			TT_01_01													:= m01_rs3_r3._01_TT_01,
			TT_01_01_offset												:= m01_rs3_r3.cart01_front_temp_offset,
			TT_01_01_error												:= m01_rs3_r3._01_TT_01_Error,
			TT_01_03													:= m01_rs3_r3._01_TT_03,               
			TT_01_03_offset												:= m01_rs3_r3.cart01_front_temp_offset,
			TT_01_03_error												:= m01_rs3_r3._01_TT_03_Error,         
			TT_02_01													:= m01_rs3_r3._02_TT_01,               
			TT_02_01_offset												:= m01_rs3_r3.cart02_front_temp_offset,
			TT_02_01_error												:= m01_rs3_r3._02_TT_01_Error,         
			TT_02_03													:= m01_rs3_r3._02_TT_03,               
			TT_02_03_offset												:= m01_rs3_r3.cart02_front_temp_offset,
			TT_02_03_error												:= m01_rs3_r3._02_TT_03_Error,         
			TT_03_01													:= m01_rs3_r3._03_TT_01,               
			TT_03_01_offset												:= m01_rs3_r3.cart03_front_temp_offset,
			TT_03_01_error												:= m01_rs3_r3._03_TT_01_Error,         
			TT_03_03													:= m01_rs3_r3._03_TT_03,               
			TT_03_03_offset												:= m01_rs3_r3.cart03_front_temp_offset,
			TT_03_03_error												:= m01_rs3_r3._03_TT_03_Error,         
			TT_04_01													:= m01_rs3_r3._04_TT_01,               
			TT_04_01_offset												:= m01_rs3_r3.cart04_front_temp_offset,
			TT_04_01_error												:= m01_rs3_r3._04_TT_01_Error,         
			TT_04_03													:= m01_rs3_r3._04_TT_03,               
			TT_04_03_offset												:= m01_rs3_r3.cart04_front_temp_offset,
			TT_04_03_error												:= m01_rs3_r3._04_TT_03_Error,         
			TT_05_01													:= m01_rs3_r3._05_TT_01,               
			TT_05_01_offset												:= m01_rs3_r3.cart05_front_temp_offset,
			TT_05_01_error												:= m01_rs3_r3._05_TT_01_Error,         
			TT_05_03													:= m01_rs3_r3._05_TT_03,               
			TT_05_03_offset												:= m01_rs3_r3.cart05_front_temp_offset,
			TT_05_03_error												:= m01_rs3_r3._05_TT_03_Error,         
			TT_06_01													:= m01_rs3_r3._06_TT_01,               
			TT_06_01_offset												:= m01_rs3_r3.cart06_front_temp_offset,
			TT_06_01_error												:= m01_rs3_r3._06_TT_01_Error,         
			TT_06_03													:= m01_rs3_r3._06_TT_03,               
			TT_06_03_offset												:= m01_rs3_r3.cart06_front_temp_offset,
			TT_06_03_error												:= m01_rs3_r3._06_TT_03_Error,         
			TT_07_01													:= m01_rs3_r3._07_TT_01,               
			TT_07_01_offset												:= m01_rs3_r3.cart07_front_temp_offset,
			TT_07_01_error												:= m01_rs3_r3._07_TT_01_Error,         
			TT_07_03													:= m01_rs3_r3._07_TT_03,               
			TT_07_03_offset												:= m01_rs3_r3.cart07_front_temp_offset,
			TT_07_03_error												:= m01_rs3_r3._07_TT_03_Error,         
			TT_08_01													:= m01_rs3_r3._08_TT_01,               
			TT_08_01_offset												:= m01_rs3_r3.cart08_front_temp_offset,
			TT_08_01_error												:= m01_rs3_r3._08_TT_01_Error,         
			TT_08_03													:= m01_rs3_r3._08_TT_03,               
			TT_08_03_offset												:= m01_rs3_r3.cart08_front_temp_offset,
			TT_08_03_error												:= m01_rs3_r3._08_TT_03_Error,         
			TT_09_01													:= m01_rs3_r3._09_TT_01,               
			TT_09_01_offset												:= m01_rs3_r3.cart09_front_temp_offset,
			TT_09_01_error												:= m01_rs3_r3._09_TT_01_Error,         
			TT_09_03													:= m01_rs3_r3._09_TT_03,               
			TT_09_03_offset												:= m01_rs3_r3.cart09_front_temp_offset,
			TT_09_03_error												:= m01_rs3_r3._09_TT_03_Error,         
			TT_10_01													:= m01_rs3_r3._10_TT_01,               
			TT_10_01_offset												:= m01_rs3_r3.cart10_front_temp_offset,
			TT_10_01_error												:= m01_rs3_r3._10_TT_01_Error,         
			TT_10_03													:= m01_rs3_r3._10_TT_03,               
			TT_10_03_offset												:= m01_rs3_r3.cart10_front_temp_offset,
			TT_10_03_error												:= m01_rs3_r3._10_TT_03_Error,         
			TT_11_01													:= m01_rs3_r3._11_TT_01,               
			TT_11_01_offset												:= m01_rs3_r3.cart11_front_temp_offset,
			TT_11_01_error												:= m01_rs3_r3._11_TT_01_Error,         
			TT_11_03													:= m01_rs3_r3._11_TT_03,               
			TT_11_03_offset												:= m01_rs3_r3.cart11_front_temp_offset,
			TT_11_03_error												:= m01_rs3_r3._11_TT_03_Error,         
			TT_12_01													:= m01_rs3_r3._12_TT_01,               
			TT_12_01_offset												:= m01_rs3_r3.cart12_front_temp_offset,
			TT_12_01_error												:= m01_rs3_r3._12_TT_01_Error,         
			TT_12_03													:= m01_rs3_r3._12_TT_03,               
			TT_12_03_offset												:= m01_rs3_r3.cart12_front_temp_offset,
			TT_12_03_error												:= m01_rs3_r3._12_TT_03_Error,         
		    
			cart01_front_temp											=> m01_rs3_r3.cart01_front_temp,						
			cart01_front_temp_error 									=> m01_rs3_r3.cart01_front_temp_error,
			cart01_back_temp											=> m01_rs3_r3.cart01_back_temp,
			cart01_back_temp_error 										=> m01_rs3_r3.cart01_back_temp_error,
			cart02_front_temp											=> m01_rs3_r3.cart02_front_temp,						
			cart02_front_temp_error 									=> m01_rs3_r3.cart02_front_temp_error,
			cart02_back_temp											=> m01_rs3_r3.cart02_back_temp,
			cart02_back_temp_error 										=> m01_rs3_r3.cart02_back_temp_error,
			cart03_front_temp											=> m01_rs3_r3.cart03_front_temp,						
			cart03_front_temp_error 									=> m01_rs3_r3.cart03_front_temp_error,
			cart03_back_temp											=> m01_rs3_r3.cart03_back_temp,
			cart03_back_temp_error 										=> m01_rs3_r3.cart03_back_temp_error,
			cart04_front_temp											=> m01_rs3_r3.cart04_front_temp,						
			cart04_front_temp_error 									=> m01_rs3_r3.cart04_front_temp_error,
			cart04_back_temp											=> m01_rs3_r3.cart04_back_temp,
			cart04_back_temp_error 										=> m01_rs3_r3.cart04_back_temp_error,
			cart05_front_temp											=> m01_rs3_r3.cart05_front_temp,						
			cart05_front_temp_error 									=> m01_rs3_r3.cart05_front_temp_error,
			cart05_back_temp											=> m01_rs3_r3.cart05_back_temp,
			cart05_back_temp_error 										=> m01_rs3_r3.cart05_back_temp_error,
			cart06_front_temp											=> m01_rs3_r3.cart06_front_temp,						
			cart06_front_temp_error 									=> m01_rs3_r3.cart06_front_temp_error,
			cart06_back_temp											=> m01_rs3_r3.cart06_back_temp,
			cart06_back_temp_error 										=> m01_rs3_r3.cart06_back_temp_error,
			cart07_front_temp											=> m01_rs3_r3.cart07_front_temp,						
			cart07_front_temp_error 									=> m01_rs3_r3.cart07_front_temp_error,
			cart07_back_temp											=> m01_rs3_r3.cart07_back_temp,
			cart07_back_temp_error 										=> m01_rs3_r3.cart07_back_temp_error,
			cart08_front_temp											=> m01_rs3_r3.cart08_front_temp,						
			cart08_front_temp_error 									=> m01_rs3_r3.cart08_front_temp_error,
			cart08_back_temp											=> m01_rs3_r3.cart08_back_temp,
			cart08_back_temp_error 										=> m01_rs3_r3.cart08_back_temp_error,
			cart09_front_temp											=> m01_rs3_r3.cart09_front_temp,						
			cart09_front_temp_error 									=> m01_rs3_r3.cart09_front_temp_error,
			cart09_back_temp											=> m01_rs3_r3.cart09_back_temp,
			cart09_back_temp_error 										=> m01_rs3_r3.cart09_back_temp_error,
			cart10_front_temp											=> m01_rs3_r3.cart10_front_temp,						
			cart10_front_temp_error 									=> m01_rs3_r3.cart10_front_temp_error,
			cart10_back_temp											=> m01_rs3_r3.cart10_back_temp,
			cart10_back_temp_error 										=> m01_rs3_r3.cart10_back_temp_error,
			cart11_front_temp											=> m01_rs3_r3.cart11_front_temp,						
			cart11_front_temp_error 									=> m01_rs3_r3.cart11_front_temp_error,
			cart11_back_temp											=> m01_rs3_r3.cart11_back_temp,
			cart11_back_temp_error 										=> m01_rs3_r3.cart11_back_temp_error,
			cart12_front_temp											=> m01_rs3_r3.cart12_front_temp,						
			cart12_front_temp_error 									=> m01_rs3_r3.cart12_front_temp_error,
			cart12_back_temp											=> m01_rs3_r3.cart12_back_temp,
			cart12_back_temp_error 										=> m01_rs3_r3.cart12_back_temp_error,    
                                                    
			inlet_co2_pump												:= m01_rs3_r3.inlet_co2_pump,
			AT_01_pump													=> m01_rs3_r3.AT_01_pump,
			inlet_co2_pump_cmd_status									=> m01_rs3_r3.inlet_co2_pump_cmd_status,
			inlet_co2_sol												:= m01_rs3_r3.inlet_co2_sol,
			AT_01_sol													=> m01_rs3_r3.AT_01_sol,
			inlet_co2_sol_cmd_status									=> m01_rs3_r3.inlet_co2_sol_cmd_status,
			outlet_co2_pump												:= m01_rs3_r3.outlet_co2_pump,
			AT_03_pump													=> m01_rs3_r3.AT_03_pump,
			outlet_co2_pump_cmd_status									=> m01_rs3_r3.outlet_co2_pump_cmd_status,
			outlet_co2_sol												:= m01_rs3_r3.outlet_co2_sol,
			AT_03_sol													=> m01_rs3_r3.AT_03_sol,
			outlet_co2_sol_cmd_status									=> m01_rs3_r3.outlet_co2_sol_cmd_status,
			repres_valve												:= m01_rs3_r3.repres_valve,
			XV_02														=> m01_rs3_r3.XV_02,
			repres_valve_open_cmd_status								=> m01_rs3_r3.repres_valve_open_cmd_status,
			repres_valve_open											:= m01_rs3_r3.repres_valve_open,
			repres_valve_closed											:= m01_rs3_r3.repres_valve_closed,
    	                                                        
			fan_vfd_control												=> m01_rs3_r3.fan_vfd_control,  		
			fan_vfd_target_vel	 		                                => m01_rs3_r3.fan_vfd_target_vel, 
			fan_vfd_enabled	 		                                    => m01_rs3_r3.fan_vfd_enabled, 
			fan_vfd_error		                                        => m01_rs3_r3.fan_vfd_error,
			fan_vfd_output												=> m01_rs3_r3.fan_vfd_output,
			fan_vfd_reset												:= m01_rs3_r3.fan_vfd_reset,
			fan_vfd_enable												:= m01_rs3_r3.fan_vfd_enable,
			fan_vfd_ecat_state											:= m01_rs3_r3.fan_vfd_ecat_state,
			fan_vfd_status												:= m01_rs3_r3.fan_vfd_status,
			fan_vfd														:= m01_rs3_r3.fan_vfd,
			fan_vfd_velocity											:= m01_rs3_r3.fan_vfd_velocity,
			fan_vfd_current												:= m01_rs3_r3.fan_vfd_current,
			fan_vfd_current_amps										=> m01_rs3_r3.fan_vfd_output_current,
			                                                    
			inlet_door_clamps_extend									:= m01_rs3_r3.inlet_door_clamps_extend,
			outlet_door_clamps_extend									:= m01_rs3_r3.outlet_door_clamps_extend,
			inlet_door_clamps_retract									:= m01_rs3_r3.inlet_door_clamps_retract,
			outlet_door_clamps_retract									:= m01_rs3_r3.outlet_door_clamps_retract,
			                                                    
			extend_clamps												:= extend_clamps,
			retract_clamps												:= retract_clamps,
			                                                    
			inlet_door_left_clamps_extend								=> m01_rs3_r3.XV_01_Left_Extend_Solenoid_Valve,
			inlet_door_right_clamps_extend								=> m01_rs3_r3.XV_01_Right_Extend_Solenoid_Valve,
			outlet_door_left_clamps_extend								=> m01_rs3_r3.XV_03_Left_Extend_Solenoid_Valve,
			outlet_door_right_clamps_extend								=> m01_rs3_r3.XV_03_Right_Extend_Solenoid_Valve,
			inlet_door_left_clamps_retract								=> m01_rs3_r3.XV_01_Left_Retract_Solenoid_Valve,
			inlet_door_right_clamps_retract								=> m01_rs3_r3.XV_01_Right_Retract_Solenoid_Valve,
			outlet_door_left_clamps_retract								=> m01_rs3_r3.XV_03_Left_Retract_Solenoid_Valve,
			outlet_door_right_clamps_retract							=> m01_rs3_r3.XV_03_Right_Retract_Solenoid_Valve,
    	                                                        
			inlet_door_left_clamps_extended								:= m01_rs3_r3.inlet_door_left_clamps_extended_ls,  
			inlet_door_right_clamps_extended							:= m01_rs3_r3.inlet_door_right_clamps_extended_ls, 
			outlet_door_left_clamps_extended							:= m01_rs3_r3.outlet_door_left_clamps_extended_ls, 
			outlet_door_right_clamps_extended							:= m01_rs3_r3.outlet_door_right_clamps_extended_ls,
			                                                    
			inlet_door_open												:= m01_rs3_r3.inlet_door_open,
			inlet_door_close											:= m01_rs3_r3.inlet_door_close,
			outlet_door_open											:= m01_rs3_r3.outlet_door_open,
			outlet_door_close											:= m01_rs3_r3.outlet_door_close,
			                                                    
			open_doors													:= open_doors,
			close_doors													:= close_doors,
			                                                    
			open_inlet_door												=> m01_rs3_r3.XV_01_Door_Open_Solenoid_Valve,
			close_inlet_door											=> m01_rs3_r3.XV_01_Door_Close_Solenoid_Valve,
			open_outlet_door											=> m01_rs3_r3.XV_03_Door_Open_Solenoid_Valve,
			close_outlet_door											=> m01_rs3_r3.XV_03_Door_Close_Solenoid_Valve,
			                                                    
			inlet_door_left_open										:= m01_rs3_r3.inlet_door_left_open_ls, 
			inlet_door_right_open										:= m01_rs3_r3.inlet_door_right_open_ls, 
			outlet_door_left_open										:= m01_rs3_r3.outlet_door_left_open_ls, 
			outlet_door_right_open										:= m01_rs3_r3.outlet_door_right_open_ls,
			inlet_door_left_closed										:= m01_rs3_r3.inlet_door_left_closed_ls, 
			inlet_door_right_closed										:= m01_rs3_r3.inlet_door_right_closed_ls, 
			outlet_door_left_closed										:= m01_rs3_r3.outlet_door_left_closed_ls, 
			outlet_door_right_closed									:= m01_rs3_r3.outlet_door_right_closed_ls,
			                                                    
			vacuum_cooling_high_temp_count								=> m01_rs3_r3.vacuum_cooling_high_temp_count,
			adsorption_high_temp_count									=> m01_rs3_r3.adsorption_high_temp_count,
			desorption_high_temp_count									=> m01_rs3_r3.desorption_air_high_temp_count);
END_ACTION

ACTION A_Reactor4_IO:
// Phase 0 - P_M01_RS03.A_Reactor4_IO
// Rev 1.0 - April 26, 2024

fb_R4_IO(	RSet														:= _RS03,
			React														:= _R4,
			
			Power_On													:= m01_rs3.power_control,
			                                                    
			sorbent_low_temp											=> m01_rs3_r4.temp_low,
			sorbent_high_temp											=> m01_rs3_r4.temp_high,
			sorbent_average_temp										=> m01_rs3_r4.temp_average,
			                                                    
			TT_01_01													:= m01_rs3_r4._01_TT_01,
			TT_01_01_offset												:= m01_rs3_r4.cart01_front_temp_offset,
			TT_01_01_error												:= m01_rs3_r4._01_TT_01_Error,
			TT_01_03													:= m01_rs3_r4._01_TT_03,               
			TT_01_03_offset												:= m01_rs3_r4.cart01_front_temp_offset,
			TT_01_03_error												:= m01_rs3_r4._01_TT_03_Error,         
			TT_02_01													:= m01_rs3_r4._02_TT_01,               
			TT_02_01_offset												:= m01_rs3_r4.cart02_front_temp_offset,
			TT_02_01_error												:= m01_rs3_r4._02_TT_01_Error,         
			TT_02_03													:= m01_rs3_r4._02_TT_03,               
			TT_02_03_offset												:= m01_rs3_r4.cart02_front_temp_offset,
			TT_02_03_error												:= m01_rs3_r4._02_TT_03_Error,         
			TT_03_01													:= m01_rs3_r4._03_TT_01,               
			TT_03_01_offset												:= m01_rs3_r4.cart03_front_temp_offset,
			TT_03_01_error												:= m01_rs3_r4._03_TT_01_Error,         
			TT_03_03													:= m01_rs3_r4._03_TT_03,               
			TT_03_03_offset												:= m01_rs3_r4.cart03_front_temp_offset,
			TT_03_03_error												:= m01_rs3_r4._03_TT_03_Error,         
			TT_04_01													:= m01_rs3_r4._04_TT_01,               
			TT_04_01_offset												:= m01_rs3_r4.cart04_front_temp_offset,
			TT_04_01_error												:= m01_rs3_r4._04_TT_01_Error,         
			TT_04_03													:= m01_rs3_r4._04_TT_03,               
			TT_04_03_offset												:= m01_rs3_r4.cart04_front_temp_offset,
			TT_04_03_error												:= m01_rs3_r4._04_TT_03_Error,         
			TT_05_01													:= m01_rs3_r4._05_TT_01,               
			TT_05_01_offset												:= m01_rs3_r4.cart05_front_temp_offset,
			TT_05_01_error												:= m01_rs3_r4._05_TT_01_Error,         
			TT_05_03													:= m01_rs3_r4._05_TT_03,               
			TT_05_03_offset												:= m01_rs3_r4.cart05_front_temp_offset,
			TT_05_03_error												:= m01_rs3_r4._05_TT_03_Error,         
			TT_06_01													:= m01_rs3_r4._06_TT_01,               
			TT_06_01_offset												:= m01_rs3_r4.cart06_front_temp_offset,
			TT_06_01_error												:= m01_rs3_r4._06_TT_01_Error,         
			TT_06_03													:= m01_rs3_r4._06_TT_03,               
			TT_06_03_offset												:= m01_rs3_r4.cart06_front_temp_offset,
			TT_06_03_error												:= m01_rs3_r4._06_TT_03_Error,         
			TT_07_01													:= m01_rs3_r4._07_TT_01,               
			TT_07_01_offset												:= m01_rs3_r4.cart07_front_temp_offset,
			TT_07_01_error												:= m01_rs3_r4._07_TT_01_Error,         
			TT_07_03													:= m01_rs3_r4._07_TT_03,               
			TT_07_03_offset												:= m01_rs3_r4.cart07_front_temp_offset,
			TT_07_03_error												:= m01_rs3_r4._07_TT_03_Error,         
			TT_08_01													:= m01_rs3_r4._08_TT_01,               
			TT_08_01_offset												:= m01_rs3_r4.cart08_front_temp_offset,
			TT_08_01_error												:= m01_rs3_r4._08_TT_01_Error,         
			TT_08_03													:= m01_rs3_r4._08_TT_03,               
			TT_08_03_offset												:= m01_rs3_r4.cart08_front_temp_offset,
			TT_08_03_error												:= m01_rs3_r4._08_TT_03_Error,         
			TT_09_01													:= m01_rs3_r4._09_TT_01,               
			TT_09_01_offset												:= m01_rs3_r4.cart09_front_temp_offset,
			TT_09_01_error												:= m01_rs3_r4._09_TT_01_Error,         
			TT_09_03													:= m01_rs3_r4._09_TT_03,               
			TT_09_03_offset												:= m01_rs3_r4.cart09_front_temp_offset,
			TT_09_03_error												:= m01_rs3_r4._09_TT_03_Error,         
			TT_10_01													:= m01_rs3_r4._10_TT_01,               
			TT_10_01_offset												:= m01_rs3_r4.cart10_front_temp_offset,
			TT_10_01_error												:= m01_rs3_r4._10_TT_01_Error,         
			TT_10_03													:= m01_rs3_r4._10_TT_03,               
			TT_10_03_offset												:= m01_rs3_r4.cart10_front_temp_offset,
			TT_10_03_error												:= m01_rs3_r4._10_TT_03_Error,         
			TT_11_01													:= m01_rs3_r4._11_TT_01,               
			TT_11_01_offset												:= m01_rs3_r4.cart11_front_temp_offset,
			TT_11_01_error												:= m01_rs3_r4._11_TT_01_Error,         
			TT_11_03													:= m01_rs3_r4._11_TT_03,               
			TT_11_03_offset												:= m01_rs3_r4.cart11_front_temp_offset,
			TT_11_03_error												:= m01_rs3_r4._11_TT_03_Error,         
			TT_12_01													:= m01_rs3_r4._12_TT_01,               
			TT_12_01_offset												:= m01_rs3_r4.cart12_front_temp_offset,
			TT_12_01_error												:= m01_rs3_r4._12_TT_01_Error,         
			TT_12_03													:= m01_rs3_r4._12_TT_03,               
			TT_12_03_offset												:= m01_rs3_r4.cart12_front_temp_offset,
			TT_12_03_error												:= m01_rs3_r4._12_TT_03_Error,         
		    
			cart01_front_temp											=> m01_rs3_r4.cart01_front_temp,						
			cart01_front_temp_error 									=> m01_rs3_r4.cart01_front_temp_error,
			cart01_back_temp											=> m01_rs3_r4.cart01_back_temp,
			cart01_back_temp_error 										=> m01_rs3_r4.cart01_back_temp_error,
			cart02_front_temp											=> m01_rs3_r4.cart02_front_temp,						
			cart02_front_temp_error 									=> m01_rs3_r4.cart02_front_temp_error,
			cart02_back_temp											=> m01_rs3_r4.cart02_back_temp,
			cart02_back_temp_error 										=> m01_rs3_r4.cart02_back_temp_error,
			cart03_front_temp											=> m01_rs3_r4.cart03_front_temp,						
			cart03_front_temp_error 									=> m01_rs3_r4.cart03_front_temp_error,
			cart03_back_temp											=> m01_rs3_r4.cart03_back_temp,
			cart03_back_temp_error 										=> m01_rs3_r4.cart03_back_temp_error,
			cart04_front_temp											=> m01_rs3_r4.cart04_front_temp,						
			cart04_front_temp_error 									=> m01_rs3_r4.cart04_front_temp_error,
			cart04_back_temp											=> m01_rs3_r4.cart04_back_temp,
			cart04_back_temp_error 										=> m01_rs3_r4.cart04_back_temp_error,
			cart05_front_temp											=> m01_rs3_r4.cart05_front_temp,						
			cart05_front_temp_error 									=> m01_rs3_r4.cart05_front_temp_error,
			cart05_back_temp											=> m01_rs3_r4.cart05_back_temp,
			cart05_back_temp_error 										=> m01_rs3_r4.cart05_back_temp_error,
			cart06_front_temp											=> m01_rs3_r4.cart06_front_temp,						
			cart06_front_temp_error 									=> m01_rs3_r4.cart06_front_temp_error,
			cart06_back_temp											=> m01_rs3_r4.cart06_back_temp,
			cart06_back_temp_error 										=> m01_rs3_r4.cart06_back_temp_error,
			cart07_front_temp											=> m01_rs3_r4.cart07_front_temp,						
			cart07_front_temp_error 									=> m01_rs3_r4.cart07_front_temp_error,
			cart07_back_temp											=> m01_rs3_r4.cart07_back_temp,
			cart07_back_temp_error 										=> m01_rs3_r4.cart07_back_temp_error,
			cart08_front_temp											=> m01_rs3_r4.cart08_front_temp,						
			cart08_front_temp_error 									=> m01_rs3_r4.cart08_front_temp_error,
			cart08_back_temp											=> m01_rs3_r4.cart08_back_temp,
			cart08_back_temp_error 										=> m01_rs3_r4.cart08_back_temp_error,
			cart09_front_temp											=> m01_rs3_r4.cart09_front_temp,						
			cart09_front_temp_error 									=> m01_rs3_r4.cart09_front_temp_error,
			cart09_back_temp											=> m01_rs3_r4.cart09_back_temp,
			cart09_back_temp_error 										=> m01_rs3_r4.cart09_back_temp_error,
			cart10_front_temp											=> m01_rs3_r4.cart10_front_temp,						
			cart10_front_temp_error 									=> m01_rs3_r4.cart10_front_temp_error,
			cart10_back_temp											=> m01_rs3_r4.cart10_back_temp,
			cart10_back_temp_error 										=> m01_rs3_r4.cart10_back_temp_error,
			cart11_front_temp											=> m01_rs3_r4.cart11_front_temp,						
			cart11_front_temp_error 									=> m01_rs3_r4.cart11_front_temp_error,
			cart11_back_temp											=> m01_rs3_r4.cart11_back_temp,
			cart11_back_temp_error 										=> m01_rs3_r4.cart11_back_temp_error,
			cart12_front_temp											=> m01_rs3_r4.cart12_front_temp,						
			cart12_front_temp_error 									=> m01_rs3_r4.cart12_front_temp_error,
			cart12_back_temp											=> m01_rs3_r4.cart12_back_temp,
			cart12_back_temp_error 										=> m01_rs3_r4.cart12_back_temp_error,  

                                                    
			inlet_co2_pump												:= m01_rs3_r4.inlet_co2_pump,
			AT_01_pump													=> m01_rs3_r4.AT_01_pump,
			inlet_co2_pump_cmd_status									=> m01_rs3_r4.inlet_co2_pump_cmd_status,
			inlet_co2_sol												:= m01_rs3_r4.inlet_co2_sol,
			AT_01_sol													=> m01_rs3_r4.AT_01_sol,
			inlet_co2_sol_cmd_status									=> m01_rs3_r4.inlet_co2_sol_cmd_status,
			outlet_co2_pump												:= m01_rs3_r4.outlet_co2_pump,
			AT_03_pump													=> m01_rs3_r4.AT_03_pump,
			outlet_co2_pump_cmd_status									=> m01_rs3_r4.outlet_co2_pump_cmd_status,
			outlet_co2_sol												:= m01_rs3_r4.outlet_co2_sol,
			AT_03_sol													=> m01_rs3_r4.AT_03_sol,
			outlet_co2_sol_cmd_status									=> m01_rs3_r4.outlet_co2_sol_cmd_status,
			repres_valve												:= m01_rs3_r4.repres_valve,
			XV_02														=> m01_rs3_r4.XV_02,
			repres_valve_open_cmd_status								=> m01_rs3_r4.repres_valve_open_cmd_status,
			repres_valve_open											:= m01_rs3_r4.repres_valve_open,
			repres_valve_closed											:= m01_rs3_r4.repres_valve_closed,
    	                                                        
			fan_vfd_control												=> m01_rs3_r4.fan_vfd_control,  		
			fan_vfd_target_vel	 		                                => m01_rs3_r4.fan_vfd_target_vel, 
			fan_vfd_enabled	 		                                    => m01_rs3_r4.fan_vfd_enabled, 
			fan_vfd_error		                                        => m01_rs3_r4.fan_vfd_error,
			fan_vfd_output												=> m01_rs3_r4.fan_vfd_output,
			fan_vfd_reset												:= m01_rs3_r4.fan_vfd_reset,
			fan_vfd_enable												:= m01_rs3_r4.fan_vfd_enable,
			fan_vfd_ecat_state											:= m01_rs3_r4.fan_vfd_ecat_state,
			fan_vfd_status												:= m01_rs3_r4.fan_vfd_status,
			fan_vfd														:= m01_rs3_r4.fan_vfd,
			fan_vfd_velocity											:= m01_rs3_r4.fan_vfd_velocity,
			fan_vfd_current												:= m01_rs3_r4.fan_vfd_current,
			fan_vfd_current_amps										=> m01_rs3_r4.fan_vfd_output_current,
			                                                    
			inlet_door_clamps_extend									:= m01_rs3_r4.inlet_door_clamps_extend,
			outlet_door_clamps_extend									:= m01_rs3_r4.outlet_door_clamps_extend,
			inlet_door_clamps_retract									:= m01_rs3_r4.inlet_door_clamps_retract,
			outlet_door_clamps_retract									:= m01_rs3_r4.outlet_door_clamps_retract,
			                                                    
			extend_clamps												:= extend_clamps,
			retract_clamps												:= retract_clamps,
			                                                    
			inlet_door_left_clamps_extend								=> m01_rs3_r4.XV_01_Left_Extend_Solenoid_Valve,
			inlet_door_right_clamps_extend								=> m01_rs3_r4.XV_01_Right_Extend_Solenoid_Valve,
			outlet_door_left_clamps_extend								=> m01_rs3_r4.XV_03_Left_Extend_Solenoid_Valve,
			outlet_door_right_clamps_extend								=> m01_rs3_r4.XV_03_Right_Extend_Solenoid_Valve,
			inlet_door_left_clamps_retract								=> m01_rs3_r4.XV_01_Left_Retract_Solenoid_Valve,
			inlet_door_right_clamps_retract								=> m01_rs3_r4.XV_01_Right_Retract_Solenoid_Valve,
			outlet_door_left_clamps_retract								=> m01_rs3_r4.XV_03_Left_Retract_Solenoid_Valve,
			outlet_door_right_clamps_retract							=> m01_rs3_r4.XV_03_Right_Retract_Solenoid_Valve,
    	                                                        
			inlet_door_left_clamps_extended								:= m01_rs3_r4.inlet_door_left_clamps_extended_ls,  
			inlet_door_right_clamps_extended							:= m01_rs3_r4.inlet_door_right_clamps_extended_ls, 
			outlet_door_left_clamps_extended							:= m01_rs3_r4.outlet_door_left_clamps_extended_ls, 
			outlet_door_right_clamps_extended							:= m01_rs3_r4.outlet_door_right_clamps_extended_ls,
			                                                    
			inlet_door_open												:= m01_rs3_r4.inlet_door_open,
			inlet_door_close											:= m01_rs3_r4.inlet_door_close,
			outlet_door_open											:= m01_rs3_r4.outlet_door_open,
			outlet_door_close											:= m01_rs3_r4.outlet_door_close,
			                                                    
			open_doors													:= open_doors,
			close_doors													:= close_doors,
			                                                    
			open_inlet_door												=> m01_rs3_r4.XV_01_Door_Open_Solenoid_Valve,
			close_inlet_door											=> m01_rs3_r4.XV_01_Door_Close_Solenoid_Valve,
			open_outlet_door											=> m01_rs3_r4.XV_03_Door_Open_Solenoid_Valve,
			close_outlet_door											=> m01_rs3_r4.XV_03_Door_Close_Solenoid_Valve,
			                                                    
			inlet_door_left_open										:= m01_rs3_r4.inlet_door_left_open_ls, 
			inlet_door_right_open										:= m01_rs3_r4.inlet_door_right_open_ls, 
			outlet_door_left_open										:= m01_rs3_r4.outlet_door_left_open_ls, 
			outlet_door_right_open										:= m01_rs3_r4.outlet_door_right_open_ls,
			inlet_door_left_closed										:= m01_rs3_r4.inlet_door_left_closed_ls, 
			inlet_door_right_closed										:= m01_rs3_r4.inlet_door_right_closed_ls, 
			outlet_door_left_closed										:= m01_rs3_r4.outlet_door_left_closed_ls, 
			outlet_door_right_closed									:= m01_rs3_r4.outlet_door_right_closed_ls,
			                                                    
			vacuum_cooling_high_temp_count								=> m01_rs3_r4.vacuum_cooling_high_temp_count,
			adsorption_high_temp_count									=> m01_rs3_r4.adsorption_high_temp_count,
			desorption_high_temp_count									=> m01_rs3_r4.desorption_air_high_temp_count);
END_ACTION

END_PROGRAM

// ---- POUs/Functions/F_HighestInt.TcPOU
FUNCTION F_HighestInt : INT
VAR_INPUT
	Value1																: INT;
	Value2																: INT;
END_VAR
VAR
END_VAR

// F_Highest2
// Rev 1.0 - March 14, 2024

F_HighestInt																:= SEL(Value1 > Value2, Value2, Value1);

END_FUNCTION

// ---- POUs/Function_Blocks/FB_ValveError.TcPOU
FUNCTION_BLOCK PUBLIC FB_ValveError
VAR_INPUT
	Command																: BOOL;
	Open																: BOOL;
	Closed																: BOOL;
END_VAR
VAR_OUTPUT
	ti_Status																: INT;
END_VAR
VAR
	Transition															: BOOL;
	tonError															: TON;
END_VAR

//// Phase 0 - FB_ValveError
//// Rev 1.0 - December 28, 2023

Transition																:= (Command AND NOT Open) OR (NOT Command AND NOT Closed);
ti_Status																	:= SEL(Transition, 0, SEL(tonError.Q, 1, 2)); 

tonError(IN:= Transition, PT:= REAL_TO_TIME(_VALVE_TIME * _SECONDS));

END_FUNCTION_BLOCK

// ---- POUs/P_Alarms_1.TcPOU
PROGRAM P_Alarms_1
VAR
	bResetAlarm															: BOOL;
	bInQueue															: BOOL;
	bClearAlarms														: BOOL;
	i																	: INT;
	iCount																: INT					:= 0;
	tonAlarmReset														: TON;
END_VAR

// Phase 0 - P_Alarms
// Rev 1.0 - February 26, 2024

bInQueue																:= m01.ts_Alarm <> '';
IF m01.ts_Alarm <> gsAlarms[0] THEN
	m01.ts_Alarm														:= gsAlarms[0];
	m01.ts_User_Message													:= gsMessages[0];
	bResetAlarm															:= m01.ts_Alarm <> '';
END_IF  

IF tonAlarmReset.Q OR (bResetAlarm AND NOT bInQueue) THEN
	bResetAlarm															:= FALSE;
	m01.tb_Alarm_Active													:= TRUE;
END_IF

IF m01.tb_Acknowledge_Alarm THEN
	m01.tb_Alarm_Active													:= FALSE;
	FOR i := 0 TO _ALARM_COUNT DO                      	    	
		gsAlarms[i] 													:= gsAlarms[i+1];
		gsMessages[i]													:= gsMessages[i+1];
	END_FOR                                 	    	
	gsAlarms[_ALARM_COUNT]												:= '';
	gsMessages[_ALARM_COUNT]											:= '';
	giAlarmCount														:= giAlarmCount - 1;
	m01.tb_Acknowledge_Alarm											:= FALSE;
END_IF                                      	    	

IF bClearAlarms THEN
	FOR i := 0 TO _ALARM_COUNT DO                      	    	
		gsAlarms[i] 													:= '';
		gsMessages[i]													:= '';
		giAlarmCount													:= 0;
		m01.tb_Alarm_Active												:= FALSE;
		bClearAlarms													:= FALSE;
	END_FOR                                 	    	
END_IF
                                            	    	
tonAlarmReset(IN:= bResetAlarm, PT:= T#1S);

METHOD M_Add_Alarm 			: BOOL
VAR_INPUT
	Unit																: STRING;
	Alarm																: STRING;
	Message																: STRING;
END_VAR
VAR
END_VAR
// Phase 0 - P_Alarms.M_Add_Alarm
// Rev 1.0 - January 31, 2024

IF giAlarmCount < _ALARM_COUNT THEN
	gsAlarms[giAlarmCount]												:= CONCAT(Unit, Alarm);
	gsMessages[giAlarmCount]											:= Message;
	giAlarmCount														:= giAlarmCount + 1;
END_IF
M_Add_Alarm																:= TRUE;
END_METHOD

METHOD M_Check_Error : BOOL
VAR_INPUT
	Error_In															: BOOL;
	Latch																: BOOL;
	Unit																: STRING;
	Alarm																: STRING;
	Message																: STRING;
END_VAR
VAR
	Error_Out															: BOOL;
END_VAR
// Phase 0 - P_Alarms.M_Check_Error
// Rev 1.0 - March 20, 2024

Error_Out																:= Latch;
IF Error_In THEN
	IF NOT Error_Out THEN
		Error_Out														:= TRUE;
		P_Alarms.M_Add_Alarm(Unit, Alarm, Message);
	END_IF
ELSE
	Error_Out															:= FALSE;
END_IF
M_Check_Error															:= Error_Out;
END_METHOD

END_PROGRAM
